TYPE DS_XMLRW :
STRUCT

	sMachineOnTime_JKS	: STRING(99);

END_STRUCT
END_TYPE

(* stored: Version 1.1.0.1, ProductVersion 3.1.4024.12
   DUT DS_XMLRW: Id {f5a731d1-d8f6-43c3-a91d-a2ebe0ecb990} *)
